{attribute 'qualified_only'}
{attribute 'strict'}
{attribute 'to_string'}
TYPE E_MESSAGE_BATCH :
(
	MSG_BATCH_NULL,
  MSG_BATCH_JOB_STARTED,
  MSG_BATCH_NEXT_IN_JOB,
  MSG_BATCH_JOB_DONE
)UINT;
END_TYPE

(* stored: Version 1.1.0.1
   DUT E_MESSAGE_BATCH: Id {819e2659-81e9-447c-9a58-b62d950558b0} *)
